PROGRAM Main1
VAR
	fbTime 		: FB_LocalSystemTime := ( bEnable := TRUE, dwCycle := 1 );
	bValid		: BOOL := FALSE;
	TimeStr		: STRING;
	
	Truck_ID			: UINT := 1;
	Trailer_ID AT %I*	: UINT;
	Lat					: STRING;
	Lon					: STRING;
	Speed				: STRING;
	EventCode			: STRING;
	Payload				: STRING;
END_VAR

(* get system time *)
WHILE bValid = FALSE DO
	fbTime(bValid => bValid);	
END_WHILE

fbTime();
TimeStr	:= SYSTEMTIME_TO_STRING(fbTime.systemTime);

(* read sensors *)
Read_FatigueCam();
Read_GPS();
Read_Payload();

(* save data to database *)

END_PROGRAM

(* stored: Version 1.1.0.1, ProductVersion 3.1.4024.6
   POU Main1: Id {d634cea7-0b2b-4450-a767-f61c97526782}, SpecialFunc None *)
